{attribute addProperty BoxType "EL3356-0030-0025"}
{attribute addProperty Id "RMB_StatusAT %I*RMB_Status_7F71BA301620RMB_Value_INT32AT %I*RMB_Value_INT_1F5759573240RMB_ControlAT %Q*RMB_Control_D468E5481620WcStateAT %I*WcState_F855686C1620InfoDataAT %I*InfoData_BC63D37F80100"}
{attribute addProperty CRC "2026441263"}
{attribute addProperty SizeInBites "160"}
{attribute addProperty SizeInBytes "20"}
TYPE EL3356_CA56400F :
STRUCT
	{attribute addProperty Name "RMB_Status"}
	RMB_Status : RMB_Status_7F71BA30;
	{attribute addProperty Name "RMB_Value_INT32"}
	RMB_Value_INT32 : RMB_Value_INT_1F575957;
	{attribute addProperty Name "RMB_Control"}
	RMB_Control : RMB_Control_D468E548;
	{attribute addProperty Name "WcState"}
	WcState : WcState_F855686C;
	{attribute addProperty Name "InfoData"}
	InfoData : InfoData_BC63D37F;
END_STRUCT
END_TYPE

(* stored: Version 1.2.0.0, ProductVersion 3.1.4024.9
   DUT EL3356_CA56400F: Id {9423bd7c-4442-4bd4-b43c-e00250d8767b} *)
